LIN {X 0,Y 62.563,Z 497.336,A -85,B 0,C 180,E1 -29428.674,E2 -29428.674} C_VEL
LIN {X 0,Y 56.7,Z 507.373,A -85,B 0,C 180,E1 -29437.429,E2 -29437.429} C_VEL
LIN {X 0,Y 52.473,Z 514.882,A -85,B 0,C 180,E1 -29446.946,E2 -29446.946} C_VEL
LIN {X 0,Y 49.586,Z 521.016,A -85,B 0,C 180,E1 -29457.713,E2 -29457.713} C_VEL
LIN {X 0,Y 48.121,Z 525.928,A -85,B 0,C 180,E1 -29469.173,E2 -29469.173} C_VEL
LIN {X 0,Y 48.879,Z 531.089,A -85,B 0,C 180,E1 -29484.892,E2 -29484.892} C_VEL
LIN {X 0,Y 52.714,Z 534.657,A -85,B 0,C 180,E1 -29498.941,E2 -29498.941} C_VEL
LIN {X 0,Y 53.805,Z 535.166,A -85,B 0,C 180,E1 -29501.479,E2 -29501.479} C_VEL
LIN {X 0,Y 56.001,Z 536.249,A -85,B 0,C 180,E1 -29507.097,E2 -29507.097} C_VEL
LIN {X 0,Y 59.2,Z 537.488,A -85,B 0,C 180,E1 -29516.359,E2 -29516.359} C_VEL
LIN {X 0,Y 63.8,Z 538.239,A -85,B 0,C 180,E1 -29524.53,E2 -29524.53} C_VEL
LIN {X 0,Y 67.91,Z 538.362,A -85,B 0,C 180,E1 -29528.221,E2 -29528.221} C_VEL
LIN {X 0,Y 72.829,Z 538.347,A -85,B 0,C 180,E1 -29531.128,E2 -29531.128} C_VEL
LIN {X 0,Y 81.161,Z 537.679,A -85,B 0,C 180,E1 -29535.057,E2 -29535.057} C_VEL
LIN {X 0,Y 93.624,Z 535.537,A -85,B 0,C 180,E1 -29539.315,E2 -29539.315} C_VEL
LIN {X 0,Y 94.286,Z 535.405,A -85,B 0,C 180,E1 -29540.065,E2 -29540.065} C_VEL
LIN {X 0,Y 92.698,Z 535.887,A -85,B 0,C 180,E1 -29541.338,E2 -29541.338} C_VEL
LIN {X 0,Y 84.567,Z 537.633,A -85,B 0,C 180,E1 -29543.918,E2 -29543.918} C_VEL
LIN {X 0,Y 72.499,Z 539.277,A -85,B 0,C 180,E1 -29549.261,E2 -29549.261} C_VEL
LIN {X 0,Y 61.355,Z 539.6,A -85,B 0,C 180,E1 -29556.7,E2 -29556.7} C_VEL
LIN {X 0,Y 51.809,Z 538.557,A -85,B 0,C 180,E1 -29567.296,E2 -29567.296} C_VEL
LIN {X 0,Y 45.145,Z 536.22,A -85,B 0,C 180,E1 -29582.163,E2 -29582.163} C_VEL
LIN {X 0,Y 42.187,Z 532.421,A -85,B 0,C 180,E1 -29600.414,E2 -29600.414} C_VEL
LIN {X 0,Y 42.067,Z 529.834,A -85,B 0,C 180,E1 -29610.004,E2 -29610.004} C_VEL
LIN {X 0,Y 42.559,Z 524.811,A -85,B 0,C 180,E1 -29624.345,E2 -29624.345} C_VEL
LIN {X 0,Y 45.941,Z 517.263,A -85,B 0,C 180,E1 -29639.817,E2 -29639.817} C_VEL
LIN {X 0,Y 50.954,Z 509.07,A -85,B 0,C 180,E1 -29650.936,E2 -29650.936} C_VEL
LIN {X 0,Y 56.276,Z 500.68,A -85,B 0,C 180,E1 -29658.534,E2 -29658.534} C_VEL
LIN {X 0,Y 57.068,Z 499.138,A -85,B 0,C 180,E1 -29659.733,E2 -29659.733} C_VEL
LIN {X 0,Y 60.113,Z 488.746,A -85,B 0,C 180,E1 -29667.849,E2 -29667.849} C_VEL
LIN {X 0,Y 61.826,Z 481.876,A -85,B 0,C 180,E1 -29672.331,E2 -29672.331} C_VEL
LIN {X 0,Y 61.553,Z 477.121,A -85,B 0,C 180,E1 -29676.441,E2 -29676.441} C_VEL
LIN {X 0,Y 60.368,Z 472.755,A -85,B 0,C 180,E1 -29681.327,E2 -29681.327} C_VEL
LIN {X 0,Y 58.713,Z 467.928,A -85,B 0,C 180,E1 -29687.808,E2 -29687.808} C_VEL
LIN {X 0,Y 57.474,Z 464.636,A -85,B 0,C 180,E1 -29692.976,E2 -29692.976} C_VEL
LIN {X 0,Y 56.105,Z 461.048,A -85,B 0,C 180,E1 -29700,E2 -29700} C_VEL
LIN {X 0,Y 54.079,Z 457.449,A -85,B 0,C 180,E1 -29715.065,E2 -29715.065} C_VEL
LIN {X 0,Y 53.674,Z 457.552,A -85,B 0,C 180,E1 -29723.565,E2 -29723.565} C_VEL
LIN {X 0,Y 53.749,Z 458.691,A -85,B 0,C 180,E1 -29731.535,E2 -29731.535} C_VEL
LIN {X 0,Y 55.481,Z 461.149,A -85,B 0,C 180,E1 -29743.313,E2 -29743.313} C_VEL
LIN {X 0,Y 57.149,Z 465.018,A -85,B 0,C 180,E1 -29752.054,E2 -29752.054} C_VEL
LIN {X 0,Y 58.939,Z 469.565,A -85,B 0,C 180,E1 -29759.482,E2 -29759.482} C_VEL
LIN {X 0,Y 60.647,Z 474.193,A -85,B 0,C 180,E1 -29765.892,E2 -29765.892} C_VEL
LIN {X 0,Y 62.357,Z 480.803,A -85,B 0,C 180,E1 -29773.291,E2 -29773.291} C_VEL
LIN {X 0,Y 62.525,Z 483.375,A -85,B 0,C 180,E1 -29775.678,E2 -29775.678} C_VEL
LIN {X 0,Y 61.372,Z 489.261,A -85,B 0,C 180,E1 -29780.107,E2 -29780.107} C_VEL
LIN {X 0,Y 54.976,Z 499.666,A -85,B 0,C 180,E1 -29787.024,E2 -29787.024} C_VEL
LIN {X 0,Y 48.938,Z 509.199,A -85,B 0,C 180,E1 -29796.782,E2 -29796.782} C_VEL
LIN {X 0,Y 44.448,Z 516.719,A -85,B 0,C 180,E1 -29808.432,E2 -29808.432} C_VEL
LIN {X 0,Y 41.635,Z 522.995,A -85,B 0,C 180,E1 -29822.435,E2 -29822.435} C_VEL
LIN {X 0,Y 41.331,Z 529.113,A -85,B 0,C 180,E1 -29841.37,E2 -29841.37} C_VEL
LIN {X 0,Y 43.638,Z 532.492,A -85,B 0,C 180,E1 -29854.621,E2 -29854.621} C_VEL
LIN {X 0,Y 49.98,Z 535.88,A -85,B 0,C 180,E1 -29869.82,E2 -29869.82} C_VEL
LIN {X 0,Y 57.793,Z 537.684,A -85,B 0,C 180,E1 -29880,E2 -29880} C_VEL
LIN {X 0,Y 67.91,Z 538.362,A -85,B 0,C 180,E1 -29888.221,E2 -29888.221} C_VEL
LIN {X 0,Y 69.187,Z 538.449,A -85,B 0,C 180,E1 -29889.85,E2 -29889.85} C_VEL
LIN {X 0,Y 69.521,Z 538.577,A -85,B 0,C 180,E1 -29892.534,E2 -29892.534} C_VEL
LIN {X 0,Y 68.525,Z 538.803,A -85,B 0,C 180,E1 -29896.192,E2 -29896.192} C_VEL
LIN {X 0,Y 67.018,Z 538.969,A -85,B 0,C 180,E1 -29899.045,E2 -29899.045} C_VEL
LIN {X 0,Y 63.515,Z 539.199,A -85,B 0,C 180,E1 -29904.078,E2 -29904.078} C_VEL
LIN {X 0,Y 59.408,Z 539.247,A -85,B 0,C 180,E1 -29908.973,E2 -29908.973} C_VEL
LIN {X 0,Y 56.163,Z 539.057,A -85,B 0,C 180,E1 -29911.941,E2 -29911.941} C_VEL
LIN {X 0,Y 46.841,Z 537.902,A -85,B 0,C 180,E1 -29921.398,E2 -29921.398} C_VEL
LIN {X 0,Y 39.033,Z 535.333,A -85,B 0,C 180,E1 -29937.31,E2 -29937.31} C_VEL
LIN {X 0,Y 35.296,Z 531.26,A -85,B 0,C 180,E1 -29958.519,E2 -29958.519} C_VEL
LIN {X 0,Y 35.038,Z 528.555,A -85,B 0,C 180,E1 -29970.004,E2 -29970.004} C_VEL
LIN {X 0,Y 35.77,Z 523.28,A -85,B 0,C 180,E1 -29987.145,E2 -29987.145} C_VEL
LIN {X 0,Y 39.161,Z 516.645,A -85,B 0,C 180,E1 -30002.579,E2 -30002.579} C_VEL
LIN {X 0,Y 44.746,Z 508.353,A -85,B 0,C 180,E1 -30014.979,E2 -30014.979} C_VEL
LIN {X 0,Y 50.585,Z 499.88,A -85,B 0,C 180,E1 -30023.028,E2 -30023.028} C_VEL
LIN {X 0,Y 53.892,Z 490.747,A -85,B 0,C 180,E1 -30030.965,E2 -30030.965} C_VEL
LIN {X 0,Y 55.955,Z 484.426,A -85,B 0,C 180,E1 -30035.586,E2 -30035.586} C_VEL
LIN {X 0,Y 56.112,Z 481.898,A -85,B 0,C 180,E1 -30037.929,E2 -30037.929} C_VEL
LIN {X 0,Y 55.85,Z 479.027,A -85,B 0,C 180,E1 -30041.188,E2 -30041.188} C_VEL
LIN {X 0,Y 54.476,Z 473.688,A -85,B 0,C 180,E1 -30048.841,E2 -30048.841} C_VEL
LIN {X 0,Y 53.239,Z 469.573,A -85,B 0,C 180,E1 -30056.215,E2 -30056.215} C_VEL
LIN {X 0,Y 52.76,Z 467.815,A -85,B 0,C 180,E1 -30059.999,E2 -30059.999} C_VEL
LIN {X 0,Y 52.214,Z 466.516,A -85,B 0,C 180,E1 -30063.858,E2 -30063.858} C_VEL
LIN {X 0,Y 51.125,Z 463.954,A -85,B 0,C 180,E1 -30075.958,E2 -30075.958} C_VEL
LIN {X 0,Y 50.719,Z 464.266,A -85,B 0,C 180,E1 -30084.563,E2 -30084.563} C_VEL
LIN {X 0,Y 50.895,Z 465.722,A -85,B 0,C 180,E1 -30094.048,E2 -30094.048} C_VEL
LIN {X 0,Y 52.003,Z 467.504,A -85,B 0,C 180,E1 -30102.51,E2 -30102.51} C_VEL
LIN {X 0,Y 53.37,Z 471.585,A -85,B 0,C 180,E1 -30112.195,E2 -30112.195} C_VEL
LIN {X 0,Y 54.978,Z 476.741,A -85,B 0,C 180,E1 -30121.098,E2 -30121.098} C_VEL
LIN {X 0,Y 56.128,Z 481.666,A -85,B 0,C 180,E1 -30127.933,E2 -30127.933} C_VEL
LIN {X 0,Y 56.663,Z 484.753,A -85,B 0,C 180,E1 -30131.743,E2 -30131.743} C_VEL
LIN {X 0,Y 55.843,Z 488.924,A -85,B 0,C 180,E1 -30135.419,E2 -30135.419} C_VEL
LIN {X 0,Y 52.835,Z 493.907,A -85,B 0,C 180,E1 -30138.488,E2 -30138.488} C_VEL
LIN {X 0,Y 46.821,Z 502.765,A -85,B 0,C 180,E1 -30145.688,E2 -30145.688} C_VEL
LIN {X 0,Y 40.886,Z 511.251,A -85,B 0,C 180,E1 -30156.409,E2 -30156.409} C_VEL
LIN {X 0,Y 36.542,Z 518.284,A -85,B 0,C 180,E1 -30170.157,E2 -30170.157} C_VEL
LIN {X 0,Y 34.015,Z 524.532,A -85,B 0,C 180,E1 -30188.299,E2 -30188.299} C_VEL
LIN {X 0,Y 34.512,Z 528.776,A -85,B 0,C 180,E1 -30204.535,E2 -30204.535} C_VEL
LIN {X 0,Y 39.384,Z 533.52,A -85,B 0,C 180,E1 -30225.279,E2 -30225.279} C_VEL
LIN {X 0,Y 47.932,Z 536.631,A -85,B 0,C 180,E1 -30240.001,E2 -30240.001} C_VEL
LIN {X 0,Y 56.867,Z 538.17,A -85,B 0,C 180,E1 -30248.644,E2 -30248.644} C_VEL
LIN {X 0,Y 65.193,Z 538.731,A -85,B 0,C 180,E1 -30254.026,E2 -30254.026} C_VEL
LIN {X 0,Y 78.448,Z 538.206,A -85,B 0,C 180,E1 -30259.77,E2 -30259.77} C_VEL
LIN {X 0,Y 75.55,Z 538.611,A -85,B 0,C 180,E1 -30261.533,E2 -30261.533} C_VEL
LIN {X 0,Y 63.264,Z 539.304,A -85,B 0,C 180,E1 -30267.292,E2 -30267.292} C_VEL
LIN {X 0,Y 56.163,Z 539.057,A -85,B 0,C 180,E1 -30271.941,E2 -30271.941} C_VEL
LIN {X 0,Y 51.248,Z 538.625,A -85,B 0,C 180,E1 -30275.378,E2 -30275.378} C_VEL
LIN {X 0,Y 42.595,Z 537.1,A -85,B 0,C 180,E1 -30280.97,E2 -30280.97} C_VEL
LIN {X 0,Y 36.095,Z 535.342,A -85,B 0,C 180,E1 -30287.136,E2 -30287.136} C_VEL
LIN {X 0,Y 32.229,Z 533.787,A -85,B 0,C 180,E1 -30294.205,E2 -30294.205} C_VEL
LIN {X 0,Y 31.288,Z 533.188,A -85,B 0,C 180,E1 -30297.191,E2 -30297.191} C_VEL
LIN {X 0,Y 28.477,Z 530.042,A -85,B 0,C 180,E1 -30315.718,E2 -30315.718} C_VEL
LIN {X 0,Y 28.009,Z 527.191,A -85,B 0,C 180,E1 -30330.005,E2 -30330.005} C_VEL
LIN {X 0,Y 29.111,Z 521.668,A -85,B 0,C 180,E1 -30351.236,E2 -30351.236} C_VEL
LIN {X 0,Y 33.456,Z 514.733,A -85,B 0,C 180,E1 -30369.07,E2 -30369.07} C_VEL
LIN {X 0,Y 40.083,Z 506.079,A -85,B 0,C 180,E1 -30382.1,E2 -30382.1} C_VEL
LIN {X 0,Y 45.203,Z 499.024,A -85,B 0,C 180,E1 -30388.779,E2 -30388.779} C_VEL
LIN {X 0,Y 49.177,Z 489.508,A -85,B 0,C 180,E1 -30397.547,E2 -30397.547} C_VEL
LIN {X 0,Y 50.58,Z 485.582,A -85,B 0,C 180,E1 -30400.731,E2 -30400.731} C_VEL
LIN {X 0,Y 50.592,Z 483.085,A -85,B 0,C 180,E1 -30403.869,E2 -30403.869} C_VEL
LIN {X 0,Y 49.737,Z 478.24,A -85,B 0,C 180,E1 -30411.876,E2 -30411.876} C_VEL
LIN {X 0,Y 48.999,Z 474.352,A -85,B 0,C 180,E1 -30419.999,E2 -30419.999} C_VEL
LIN {X 0,Y 48.676,Z 472.858,A -85,B 0,C 180,E1 -30424.139,E2 -30424.139} C_VEL
LIN {X 0,Y 48.241,Z 471.8,A -85,B 0,C 180,E1 -30428.376,E2 -30428.376} C_VEL
LIN {X 0,Y 47.818,Z 470.339,A -85,B 0,C 180,E1 -30437.094,E2 -30437.094} C_VEL
LIN {X 0,Y 47.364,Z 471.055,A -85,B 0,C 180,E1 -30447.084,E2 -30447.084} C_VEL
LIN {X 0,Y 47.668,Z 472.452,A -85,B 0,C 180,E1 -30456.138,E2 -30456.138} C_VEL
LIN {X 0,Y 48.275,Z 474.285,A -85,B 0,C 180,E1 -30463.285,E2 -30463.285} C_VEL
LIN {X 0,Y 49.007,Z 476.952,A -85,B 0,C 180,E1 -30470.328,E2 -30470.328} C_VEL
LIN {X 0,Y 50.064,Z 481.864,A -85,B 0,C 180,E1 -30479.889,E2 -30479.889} C_VEL
LIN {X 0,Y 50.751,Z 487.025,A -85,B 0,C 180,E1 -30487.715,E2 -30487.715} C_VEL
LIN {X 0,Y 50.24,Z 489.853,A -85,B 0,C 180,E1 -30490.746,E2 -30490.746} C_VEL
LIN {X 0,Y 43.186,Z 499.699,A -85,B 0,C 180,E1 -30497.531,E2 -30497.531} C_VEL
LIN {X 0,Y 36.662,Z 508.191,A -85,B 0,C 180,E1 -30507.249,E2 -30507.249} C_VEL
LIN {X 0,Y 30.551,Z 516.436,A -85,B 0,C 180,E1 -30523.294,E2 -30523.294} C_VEL
LIN {X 0,Y 27.486,Z 521.993,A -85,B 0,C 180,E1 -30540.75,E2 -30540.75} C_VEL
LIN {X 0,Y 27.05,Z 526.751,A -85,B 0,C 180,E1 -30561.201,E2 -30561.201} C_VEL
LIN {X 0,Y 29.838,Z 530.699,A -85,B 0,C 180,E1 -30580.4,E2 -30580.4} C_VEL
LIN {X 0,Y 38.021,Z 534.884,A -85,B 0,C 180,E1 -30600.001,E2 -30600.001} C_VEL
LIN {X 0,Y 45.412,Z 536.915,A -85,B 0,C 180,E1 -30608.904,E2 -30608.904} C_VEL
LIN {X 0,Y 53.551,Z 538.283,A -85,B 0,C 180,E1 -30615.218,E2 -30615.218} C_VEL
LIN {X 0,Y 62.178,Z 538.951,A -85,B 0,C 180,E1 -30619.822,E2 -30619.822} C_VEL
LIN {X 0,Y 60.331,Z 538.973,A -85,B 0,C 180,E1 -30621.272,E2 -30621.272} C_VEL
LIN {X 0,Y 48.108,Z 538.117,A -85,B 0,C 180,E1 -30628.78,E2 -30628.78} C_VEL
LIN {X 0,Y 37.461,Z 535.93,A -85,B 0,C 180,E1 -30641.378,E2 -30641.378} C_VEL
LIN {X 0,Y 31.288,Z 533.188,A -85,B 0,C 180,E1 -30657.191,E2 -30657.191} C_VEL
LIN {X 0,Y 28.601,Z 531.402,A -85,B 0,C 180,E1 -30666.631,E2 -30666.631} C_VEL
LIN {X 0,Y 25.812,Z 529.163,A -85,B 0,C 180,E1 -30676.683,E2 -30676.683} C_VEL
LIN {X 0,Y 22.05,Z 523.727,A -85,B 0,C 180,E1 -30701.258,E2 -30701.258} C_VEL
LIN {X 0,Y 22.896,Z 519.573,A -85,B 0,C 180,E1 -30718.977,E2 -30718.977} C_VEL
LIN {X 0,Y 28.337,Z 512.666,A -85,B 0,C 180,E1 -30738.084,E2 -30738.084} C_VEL
LIN {X 0,Y 34.768,Z 505.263,A -85,B 0,C 180,E1 -30749.223,E2 -30749.223} C_VEL
LIN {X 0,Y 39.051,Z 500.077,A -85,B 0,C 180,E1 -30754.146,E2 -30754.146} C_VEL
LIN {X 0,Y 41.323,Z 496.057,A -85,B 0,C 180,E1 -30758.27,E2 -30758.27} C_VEL
LIN {X 0,Y 44.669,Z 489.203,A -85,B 0,C 180,E1 -30764.515,E2 -30764.515} C_VEL
LIN {X 0,Y 45.233,Z 487.673,A -85,B 0,C 180,E1 -30766.064,E2 -30766.064} C_VEL
LIN {X 0,Y 45.14,Z 484.799,A -85,B 0,C 180,E1 -30771.042,E2 -30771.042} C_VEL
LIN {X 0,Y 44.835,Z 480.7,A -85,B 0,C 180,E1 -30779.999,E2 -30779.999} C_VEL
LIN {X 0,Y 44.704,Z 479.045,A -85,B 0,C 180,E1 -30784.508,E2 -30784.508} C_VEL
LIN {X 0,Y 44.506,Z 477.848,A -85,B 0,C 180,E1 -30789.085,E2 -30789.085} C_VEL
LIN {X 0,Y 44.238,Z 476.572,A -85,B 0,C 180,E1 -30797.585,E2 -30797.585} C_VEL
LIN {X 0,Y 43.709,Z 477.535,A -85,B 0,C 180,E1 -30808.839,E2 -30808.839} C_VEL
LIN {X 0,Y 44.001,Z 479.445,A -85,B 0,C 180,E1 -30819.709,E2 -30819.709} C_VEL
LIN {X 0,Y 44.446,Z 481.836,A -85,B 0,C 180,E1 -30827.313,E2 -30827.313} C_VEL
LIN {X 0,Y 44.932,Z 486.572,A -85,B 0,C 180,E1 -30837.968,E2 -30837.968} C_VEL
LIN {X 0,Y 44.978,Z 490.411,A -85,B 0,C 180,E1 -30844.548,E2 -30844.548} C_VEL
LIN {X 0,Y 37.001,Z 500.722,A -85,B 0,C 180,E1 -30851.749,E2 -30851.749} C_VEL
LIN {X 0,Y 29.405,Z 509.515,A -85,B 0,C 180,E1 -30862.827,E2 -30862.827} C_VEL
LIN {X 0,Y 22.883,Z 517.422,A -85,B 0,C 180,E1 -30882.409,E2 -30882.409} C_VEL
LIN {X 0,Y 19.896,Z 523.153,A -85,B 0,C 180,E1 -30907.888,E2 -30907.888} C_VEL
LIN {X 0,Y 22.265,Z 528.834,A -85,B 0,C 180,E1 -30941.601,E2 -30941.601} C_VEL
LIN {X 0,Y 28.109,Z 532.417,A -85,B 0,C 180,E1 -30960.001,E2 -30960.001} C_VEL
LIN {X 0,Y 35.858,Z 535.208,A -85,B 0,C 180,E1 -30971.508,E2 -30971.508} C_VEL
LIN {X 0,Y 44.56,Z 537.282,A -85,B 0,C 180,E1 -30978.871,E2 -30978.871} C_VEL
LIN {X 0,Y 45.126,Z 537.441,A -85,B 0,C 180,E1 -30980.872,E2 -30980.872} C_VEL
LIN {X 0,Y 33.211,Z 535.016,A -85,B 0,C 180,E1 -30992.18,E2 -30992.18} C_VEL
LIN {X 0,Y 24.158,Z 531.239,A -85,B 0,C 180,E1 -31014.428,E2 -31014.428} C_VEL
LIN {X 0,Y 21.288,Z 527.347,A -85,B 0,C 180,E1 -31040.506,E2 -31040.506} C_VEL
LIN {X 0,Y 21.057,Z 523.942,A -85,B 0,C 180,E1 -31059.614,E2 -31059.614} C_VEL
LIN {X 0,Y 22.896,Z 519.573,A -85,B 0,C 180,E1 -31078.977,E2 -31078.977} C_VEL
LIN {X 0,Y 24.651,Z 516.295,A -85,B 0,C 180,E1 -31090.05,E2 -31090.05} C_VEL
LIN {X 0,Y 27.517,Z 510.236,A -85,B 0,C 180,E1 -31106.13,E2 -31106.13} C_VEL
LIN {X 0,Y 30.56,Z 504.949,A -85,B 0,C 180,E1 -31116.354,E2 -31116.354} C_VEL
LIN {X 0,Y 34.685,Z 499.279,A -85,B 0,C 180,E1 -31123.046,E2 -31123.046} C_VEL
LIN {X 0,Y 38.698,Z 492.835,A -85,B 0,C 180,E1 -31129.535,E2 -31129.535} C_VEL
LIN {X 0,Y 39.681,Z 491.108,A -85,B 0,C 180,E1 -31131.084,E2 -31131.084} C_VEL
LIN {X 0,Y 40.086,Z 490.051,A -85,B 0,C 180,E1 -31132.443,E2 -31132.443} C_VEL
LIN {X 0,Y 40.27,Z 486.863,A -85,B 0,C 180,E1 -31139.999,E2 -31139.999} C_VEL
LIN {X 0,Y 40.347,Z 485.063,A -85,B 0,C 180,E1 -31144.996,E2 -31144.996} C_VEL
LIN {X 0,Y 40.393,Z 483.706,A -85,B 0,C 180,E1 -31150.019,E2 -31150.019} C_VEL
LIN {X 0,Y 40.068,Z 482.844,A -85,B 0,C 180,E1 -31160.536,E2 -31160.536} C_VEL
LIN {X 0,Y 39.751,Z 483.42,A -85,B 0,C 180,E1 -31167.862,E2 -31167.862} C_VEL
LIN {X 0,Y 39.717,Z 484.648,A -85,B 0,C 180,E1 -31176.318,E2 -31176.318} C_VEL
LIN {X 0,Y 39.78,Z 485.801,A -85,B 0,C 180,E1 -31181.241,E2 -31181.241} C_VEL
LIN {X 0,Y 39.716,Z 488.318,A -85,B 0,C 180,E1 -31188.713,E2 -31188.713} C_VEL
LIN {X 0,Y 39.679,Z 490.928,A -85,B 0,C 180,E1 -31195.119,E2 -31195.119} C_VEL
LIN {X 0,Y 39.487,Z 492.217,A -85,B 0,C 180,E1 -31197.724,E2 -31197.724} C_VEL
LIN {X 0,Y 31.352,Z 501.719,A -85,B 0,C 180,E1 -31203.72,E2 -31203.72} C_VEL
LIN {X 0,Y 22.745,Z 510.525,A -85,B 0,C 180,E1 -31215.1,E2 -31215.1} C_VEL
LIN {X 0,Y 15.775,Z 517.562,A -85,B 0,C 180,E1 -31236.703,E2 -31236.703} C_VEL
LIN {X 0,Y 12.78,Z 523.241,A -85,B 0,C 180,E1 -31275.199,E2 -31275.199} C_VEL
LIN {X 0,Y 18.19,Z 529.118,A -85,B 0,C 180,E1 -31320.002,E2 -31320.002} C_VEL
LIN {X 0,Y 29.86,Z 533.956,A -85,B 0,C 180,E1 -31339.72,E2 -31339.72} C_VEL
LIN {X 0,Y 30.054,Z 534.038,A -85,B 0,C 180,E1 -31340.727,E2 -31340.727} C_VEL
LIN {X 0,Y 18.913,Z 529.961,A -85,B 0,C 180,E1 -31362.009,E2 -31362.009} C_VEL
LIN {X 0,Y 14.463,Z 525.873,A -85,B 0,C 180,E1 -31395.949,E2 -31395.949} C_VEL
LIN {X 0,Y 14.567,Z 521.347,A -85,B 0,C 180,E1 -31431.224,E2 -31431.224} C_VEL
LIN {X 0,Y 20.139,Z 514.484,A -85,B 0,C 180,E1 -31461.751,E2 -31461.751} C_VEL
LIN {X 0,Y 28.635,Z 505.966,A -85,B 0,C 180,E1 -31476.994,E2 -31476.994} C_VEL
LIN {X 0,Y 34.685,Z 499.279,A -85,B 0,C 180,E1 -31483.046,E2 -31483.046} C_VEL
LIN {X 0,Y 36.137,Z 496.858,A -85,B 0,C 180,E1 -31485.942,E2 -31485.942} C_VEL
LIN {X 0,Y 36.773,Z 494.625,A -85,B 0,C 180,E1 -31489.957,E2 -31489.957} C_VEL
LIN {X 0,Y 36.89,Z 492.43,A -85,B 0,C 180,E1 -31495.548,E2 -31495.548} C_VEL
LIN {X 0,Y 36.473,Z 490.204,A -85,B 0,C 180,E1 -31504.341,E2 -31504.341} C_VEL
LIN {X 0,Y 36.02,Z 489.286,A -85,B 0,C 180,E1 -31511.341,E2 -31511.341} C_VEL
LIN {X 0,Y 35.853,Z 489.153,A -85,B 0,C 180,E1 -31513.735,E2 -31513.735} C_VEL
LIN {X 0,Y 35.669,Z 488.828,A -85,B 0,C 180,E1 -31523.207,E2 -31523.207} C_VEL
LIN {X 0,Y 35.219,Z 490.601,A -85,B 0,C 180,E1 -31537.034,E2 -31537.034} C_VEL
LIN {X 0,Y 34.767,Z 492.784,A -85,B 0,C 180,E1 -31544.898,E2 -31544.898} C_VEL
LIN {X 0,Y 34.552,Z 494.029,A -85,B 0,C 180,E1 -31548.584,E2 -31548.584} C_VEL
LIN {X 0,Y 25.608,Z 503.544,A -85,B 0,C 180,E1 -31553.126,E2 -31553.126} C_VEL
LIN {X 0,Y 15.658,Z 512.322,A -85,B 0,C 180,E1 -31563.32,E2 -31563.32} C_VEL
LIN {X 0,Y 7.098,Z 519.47,A -85,B 0,C 180,E1 -31598.071,E2 -31598.071} C_VEL
LIN {X 0,Y 9.442,Z 525.746,A -85,B 0,C 180,E1 -31686.72,E2 -31686.72} C_VEL
LIN {X 0,Y 13.991,Z 528.119,A -85,B 0,C 180,E1 -31700.337,E2 -31700.337} C_VEL
LIN {X 0,Y 11.296,Z 526.852,A -85,B 0,C 180,E1 -31714.299,E2 -31714.299} C_VEL
LIN {X 0,Y 8.239,Z 524.691,A -85,B 0,C 180,E1 -31738.552,E2 -31738.552} C_VEL
LIN {X 0,Y 7.606,Z 520.561,A -85,B 0,C 180,E1 -31797.537,E2 -31797.537} C_VEL
LIN {X 0,Y 15.151,Z 513.643,A -85,B 0,C 180,E1 -31838.109,E2 -31838.109} C_VEL
LIN {X 0,Y 24.987,Z 505.069,A -85,B 0,C 180,E1 -31849.913,E2 -31849.913} C_VEL
LIN {X 0,Y 30.943,Z 499.036,A -85,B 0,C 180,E1 -31853.593,E2 -31853.593} C_VEL
LIN {X 0,Y 35.146,Z 493.155,A -85,B 0,C 180,E1 -31859.159,E2 -31859.159} C_VEL
LIN {X 0,Y 35.603,Z 490.925,A -85,B 0,C 180,E1 -31865.663,E2 -31865.663} C_VEL
LIN {X 0,Y 35.967,Z 489.203,A -85,B 0,C 180,E1 -31872.294,E2 -31872.294} C_VEL
LIN {X 0,Y 35.853,Z 489.153,A -85,B 0,C 180,E1 -31873.735,E2 -31873.735} C_VEL
LIN {X 0,Y 35.19,Z 489.637,A -85,B 0,C 180,E1 -31877.515,E2 -31877.515} C_VEL
LIN {X 0,Y 33.673,Z 491.394,A -85,B 0,C 180,E1 -31881.811,E2 -31881.811} C_VEL
LIN {X 0,Y 30.689,Z 495.119,A -85,B 0,C 180,E1 -31889.746,E2 -31889.746} C_VEL
LIN {X 0,Y 30.266,Z 495.803,A -85,B 0,C 180,E1 -31892.854,E2 -31892.854} C_VEL
LIN {X 0,Y 30.125,Z 496.418,A -85,B 0,C 180,E1 -31897.059,E2 -31897.059} C_VEL
LIN {X 0,Y 20.773,Z 505.593,A -85,B 0,C 180,E1 -31897.196,E2 -31897.196} C_VEL
LIN {X 0,Y 10.544,Z 513.821,A -85,B 0,C 180,E1 -31895.811,E2 -31895.811} C_VEL
LIN {X 0,Y 3.805,Z 518.404,A -85,B 0,C 180,E1 -31885.033,E2 -31885.033} C_VEL
LIN {X 0,Y 5.886,Z 517.225,A -85,B 0,C 180,E1 -31864.955,E2 -31864.955} C_VEL
LIN {X 0,Y 17.657,Z 508.664,A -85,B 0,C 180,E1 -31865.594,E2 -31865.594} C_VEL
LIN {X 0,Y 26.514,Z 500.683,A -85,B 0,C 180,E1 -31866.234,E2 -31866.234} C_VEL
LIN {X 0,Y 28.293,Z 498.854,A -85,B 0,C 180,E1 -31866.446,E2 -31866.446} C_VEL
LIN {X 0,Y 29.489,Z 497.443,A -85,B 0,C 180,E1 -31867.537,E2 -31867.537} C_VEL
LIN {X 0,Y 30.78,Z 495.787,A -85,B 0,C 180,E1 -31869.541,E2 -31869.541} C_VEL
LIN {X 0,Y 31.171,Z 494.891,A -85,B 0,C 180,E1 -31873.029,E2 -31873.029} C_VEL
LIN {X 0,Y 30.904,Z 494.682,A -85,B 0,C 180,E1 -31884.531,E2 -31884.531} C_VEL
LIN {X 0,Y 30.266,Z 495.803,A -85,B 0,C 180,E1 -31892.854,E2 -31892.854} C_VEL
LIN {X 0,Y 30.154,Z 497.731,A -85,B 0,C 180,E1 -31895.627,E2 -31895.627} C_VEL
LIN {X 0,Y 30.154,Z 600,A -85,B 0,C 180,E1 -31895.627,E2 -31895.627} C_VEL
LIN {X 0,Y 30.154,Z 600,A -85,B 0,C 180,E1 -31895.627,E2 -31895.627}

QRS_NEXT_CUT()

QRS_NEXT()
QRS_HOME()

END
